(*********************************** G.D S.p.A. - Technical Department ***********************************
============= PROGRAM INFO ============
FOLDER:             TBD
MACHINES INVOLVED:  TBD 

============= DESCRIPTION =============
csp main interface program

============= REVISIONS ===============
Date		Version	 	Author      	Description             
----------	-------		------------  	--------------------------------------------
2019/09/27 	0000.00	 	M.Grasso		Creation of the PRG

**********************************************************************************************************)
PROGRAM _csp_case_transport_normal
VAR
END_VAR

(* CSP *)
	(* TRANSPORT *)
		(* ACC-U-CHANGE *)
		csp_case_transport_accU();
		(* TENSIONER *)
		csp_case_transport_tensioner();

END_PROGRAM

(* stored: Version 1.1.0.1, ProductVersion 3.1.4024.3
   POU _csp_case_transport_normal: Id {aaadf553-89fc-404e-a0c2-9ebea9dbc4bc}, SpecialFunc None *)
